# EPICS autosave request: iocs/eigerIOC/iocBoot/iocEiger1/auto_settings.req
file "eiger1_settings.req",       P=$(P),  R=cam1:
file "NDStdArrays_settings.req",  P=$(P),  R=image1:
file "NDStdArrays_settings.req",  P=$(P),  R=image2:
file "commonPlugin_settings.req", P=$(P)
